  MoveL 1561 to (-1310, 1200, 50) mm, rotated rx -180 ry 0 rz 90 deg; joints [32.484, -88.139, 132.915, -62.258, 22.45, 86.682]
  MoveL 1562 to (-1310, 1200, -0.5) mm, rotated rx -180 ry 0 rz 90 deg; joints [32.484, -85.465, 133.659, -70.1, 21.066, 95.123]
  MoveL 1563 to (-1310, 1200, 50) mm, rotated rx -180 ry 0 rz 90 deg; joints [32.484, -88.139, 132.915, -62.258, 22.45, 86.682]
  MoveL 1564 to (-1380, 11.8, 50) mm, rotated rx 180 ry 0 rz 90 deg; joints [18.052, -40.759, 62.144, -21.097, 32.805, 32.18]
  MoveL 1565 to (-1380, 11.8, -0.5) mm, rotated rx 180 ry 0 rz 90 deg; joints [18.052, -39.615, 62.725, -22.113, 31.202, 33.378]
  MoveL 1566 to (-1380, 11.8, 50) mm, rotated rx 180 ry 0 rz 90 deg; joints [18.052, -40.759, 62.144, -21.097, 32.805, 32.18]
  MoveL 1567 to (-1380, 76, 50) mm, rotated rx -180 ry 0 rz 90 deg; joints [18.556, -43.766, 67.494, -23.018, 30.808, 34.667]
  MoveL 1568 to (-1380, 76, -0.5) mm, rotated rx -180 ry 0 rz 90 deg; joints [18.556, -42.567, 68.052, -24.238, 29.198, 36.076]
  MoveL 1569 to (-1380, 76, 50) mm, rotated rx -180 ry 0 rz 90 deg; joints [18.556, -43.766, 67.494, -23.018, 30.808, 34.667]
  MoveL 1570 to (-1380, 140.2, 50) mm, rotated rx 180 ry 0 rz 90 deg; joints [19.087, -46.61, 72.487, -25.083, 29.042, 37.307]
  MoveL 1571 to (-1380, 140.2, -0.5) mm, rotated rx 180 ry 0 rz 90 deg; joints [19.087, -45.356, 73.03, -26.54, 27.424, 38.96]
  MoveL 1572 to (-1380, 140.2, 50) mm, rotated rx 180 ry 0 rz 90 deg; joints [19.087, -46.61, 72.487, -25.083, 29.042, 37.307]
  MoveL 1573 to (-1450, 11.8, 50) mm, rotated rx 180 ry 0 rz 90 deg; joints [19.677, -39.594, 60.053, -22.133, 34.225, 34.119]
  MoveL 1574 to (-1450, 11.8, -0.5) mm, rotated rx -180 ry 0 rz 90 deg; joints [19.677, -38.471, 60.644, -23.132, 32.643, 35.316]
  MoveL 1575 to (-1450, 11.8, 50) mm, rotated rx 180 ry 0 rz 90 deg; joints [19.677, -39.594, 60.053, -22.133, 34.225, 34.119]
  MoveL 1576 to (-1450, 76, 50) mm, rotated rx 180 ry 0 rz 90 deg; joints [20.219, -42.64, 65.499, -24.078, 32.216, 36.683]
  MoveL 1577 to (-1450, 76, -0.5) mm, rotated rx -180 ry 0 rz 90 deg; joints [20.219, -41.462, 66.064, -25.27, 30.631, 38.08]
  MoveL 1578 to (-1450, 76, 50) mm, rotated rx 180 ry 0 rz 90 deg; joints [20.219, -42.64, 65.499, -24.078, 32.216, 36.683]
  MoveL 1579 to (-1450, 140.2, 50) mm, rotated rx 180 ry 0 rz 90 deg; joints [20.79, -45.509, 70.561, -26.153, 30.45, 39.383]
  MoveL 1580 to (-1450, 140.2, -0.5) mm, rotated rx 180 ry 0 rz 90 deg; joints [20.79, -44.276, 71.109, -27.566, 28.861, 41.009]
  MoveL 1581 to (-1450, 140.2, 50) mm, rotated rx 180 ry 0 rz 90 deg; joints [20.79, -45.509, 70.561, -26.153, 30.45, 39.383]
  MoveL 1582 to (-1520, 53.8, 50) mm, rotated rx 180 ry 0 rz 90 deg; joints [21.645, -40.349, 61.409, -24.261, 34.398, 37.539]
  MoveL 1583 to (-1520, 53.8, -0.5) mm, rotated rx 180 ry 0 rz 90 deg; joints [21.645, -39.213, 61.993, -25.347, 32.836, 38.843]
  MoveL 1584 to (-1520, 53.8, 50) mm, rotated rx 180 ry 0 rz 90 deg; joints [21.645, -40.349, 61.409, -24.261, 34.398, 37.539]
  MoveL 1585 to (-1520, 83.81, 50) mm, rotated rx 180 ry 0 rz 90 deg; joints [21.92, -41.757, 63.927, -25.195, 33.497, 38.787]
  MoveL 1586 to (-1520, 83.81, -0.5) mm, rotated rx 180 ry 0 rz 90 deg; joints [21.92, -40.595, 64.5, -26.369, 31.935, 40.183]
  MoveL 1587 to (-1520, 83.81, 50) mm, rotated rx 180 ry 0 rz 90 deg; joints [21.92, -41.757, 63.927, -25.195, 33.497, 38.787]
  MoveL 1588 to (-1520, 129.48, 50) mm, rotated rx 180 ry 0 rz 90 deg; joints [22.352, -43.823, 67.594, -26.664, 32.23, 40.736]
  MoveL 1589 to (-1520, 129.48, -0.5) mm, rotated rx 180 ry 0 rz 90 deg; joints [22.352, -42.623, 68.152, -27.983, 30.668, 42.283]
  MoveL 1590 to (-1520, 129.48, 50) mm, rotated rx 180 ry 0 rz 90 deg; joints [22.352, -43.823, 67.594, -26.664, 32.23, 40.736]
  MoveL 1591 to (-1520, 159.49, 50) mm, rotated rx 180 ry 0 rz 90 deg; joints [22.645, -45.136, 69.907, -27.661, 31.462, 42.052]
  MoveL 1592 to (-1520, 159.49, -0.5) mm, rotated rx -180 ry 0 rz 90 deg; joints [22.645, -43.911, 70.457, -29.083, 29.9, 43.705]
  MoveL 1593 to (-1520, 159.49, 50) mm, rotated rx 180 ry 0 rz 90 deg; joints [22.645, -45.136, 69.907, -27.661, 31.462, 42.052]
  MoveL 1594 to (-1520, 205.16, 50) mm, rotated rx -180 ry 0 rz 90 deg; joints [23.105, -47.076, 73.298, -29.226, 30.384, 44.107]
  MoveL 1595 to (-1520, 205.16, -0.5) mm, rotated rx -180 ry 0 rz 90 deg; joints [23.105, -45.813, 73.839, -30.815, 28.822, 45.934]
  MoveL 1596 to (-1520, 205.16, 50) mm, rotated rx -180 ry 0 rz 90 deg; joints [23.105, -47.076, 73.298, -29.226, 30.384, 44.107]
  MoveL 1597 to (-1520, 235.17, 50) mm, rotated rx 180 ry 0 rz 90 deg; joints [23.417, -48.317, 75.451, -30.286, 29.731, 45.493]
  MoveL 1598 to (-1520, 235.17, -0.5) mm, rotated rx -180 ry 0 rz 90 deg; joints [23.417, -47.029, 75.986, -31.991, 28.169, 47.441]
  MoveL 1599 to (-1520, 235.17, 50) mm, rotated rx 180 ry 0 rz 90 deg; joints [23.417, -48.317, 75.451, -30.286, 29.731, 45.493]
  MoveL 1600 to (-1520, 280.84, 50) mm, rotated rx 180 ry 0 rz 90 deg; joints [23.907, -50.16, 78.622, -31.943, 28.818, 47.655]
  MoveL 1601 to (-1520, 280.84, -0.5) mm, rotated rx 180 ry 0 rz 90 deg; joints [23.907, -48.834, 79.152, -33.836, 27.259, 49.799]
  MoveL 1602 to (-1520, 280.84, 50) mm, rotated rx 180 ry 0 rz 90 deg; joints [23.907, -50.16, 78.622, -31.943, 28.818, 47.655]
  MoveL 1603 to (-1520, 310.85, 50) mm, rotated rx -180 ry 0 rz 90 deg; joints [24.239, -51.345, 80.643, -33.06, 28.269, 49.11]
  MoveL 1604 to (-1520, 310.85, -0.5) mm, rotated rx 180 ry 0 rz 90 deg; joints [24.239, -49.994, 81.17, -35.083, 26.713, 51.39]
  MoveL 1605 to (-1520, 310.85, 50) mm, rotated rx -180 ry 0 rz 90 deg; joints [24.239, -51.345, 80.643, -33.06, 28.269, 49.11]
  MoveL 1606 to (-1520, 356.52, 50) mm, rotated rx -180 ry 0 rz 90 deg; joints [24.762, -53.113, 83.632, -34.799, 27.509, 51.372]
  MoveL 1607 to (-1520, 356.52, -0.5) mm, rotated rx -180 ry 0 rz 90 deg; joints [24.762, -51.723, 84.157, -37.029, 25.958, 53.868]
  MoveL 1608 to (-1520, 356.52, 50) mm, rotated rx -180 ry 0 rz 90 deg; joints [24.762, -53.113, 83.632, -34.799, 27.509, 51.372]
  MoveL 1609 to (-1520, 386.53, 50) mm, rotated rx -180 ry 0 rz 90 deg; joints [25.118, -54.254, 85.543, -35.963, 27.057, 52.887]
  MoveL 1610 to (-1520, 386.53, -0.5) mm, rotated rx 180 ry 0 rz 90 deg; joints [25.118, -52.838, 86.067, -38.336, 25.511, 55.533]
  MoveL 1611 to (-1520, 386.53, 50) mm, rotated rx -180 ry 0 rz 90 deg; joints [25.118, -54.254, 85.543, -35.963, 27.057, 52.887]
  MoveL 1612 to (-1690.15, 68.53, 50) mm, rotated rx -180 ry 0 rz 90 deg; joints [25.576, -37.451, 56.183, -26.136, 38.079, 41.521]
  MoveL 1613 to (-1690.15, 68.53, -0.5) mm, rotated rx 180 ry 0 rz 90 deg; joints [25.576, -36.367, 56.797, -27.135, 36.56, 42.777]
  MoveL 1614 to (-1690.15, 68.53, 50) mm, rotated rx -180 ry 0 rz 90 deg; joints [25.576, -37.451, 56.183, -26.136, 38.079, 41.521]
  MoveL 1615 to (-1690.15, 118.53, 50) mm, rotated rx -180 ry 0 rz 90 deg; joints [26.104, -39.85, 60.513, -27.686, 36.582, 43.694]
  MoveL 1616 to (-1690.15, 118.53, -0.5) mm, rotated rx 180 ry 0 rz 90 deg; joints [26.104, -38.722, 61.101, -28.811, 35.07, 45.082]
  MoveL 1617 to (-1690.15, 118.53, 50) mm, rotated rx -180 ry 0 rz 90 deg; joints [26.104, -39.85, 60.513, -27.686, 36.582, 43.694]
  MoveL 1618 to (-1690.15, 168.53, 50) mm, rotated rx 180 ry 0 rz 90 deg; joints [26.653, -42.117, 64.568, -29.281, 35.254, 45.912]
  MoveL 1619 to (-1690.15, 168.53, -0.5) mm, rotated rx -180 ry 0 rz 90 deg; joints [26.653, -40.948, 65.138, -30.543, 33.747, 47.443]
  MoveL 1620 to (-1690.15, 168.53, 50) mm, rotated rx 180 ry 0 rz 90 deg; joints [26.653, -42.117, 64.568, -29.281, 35.254, 45.912]
  MoveL 1621 to (-1690.15, 271.33, 50) mm, rotated rx -180 ry 0 rz 90 deg; joints [27.851, -46.461, 72.228, -32.698, 32.973, 50.629]
  MoveL 1622 to (-1690.15, 271.33, -0.5) mm, rotated rx 180 ry 0 rz 90 deg; joints [27.851, -45.21, 72.771, -34.268, 31.477, 52.485]
  MoveL 1623 to (-1690.15, 271.33, 50) mm, rotated rx -180 ry 0 rz 90 deg; joints [27.851, -46.461, 72.228, -32.698, 32.973, 50.629]
  MoveL 1624 to (-1690.15, 321.33, 50) mm, rotated rx -180 ry 0 rz 90 deg; joints [28.471, -48.452, 75.685, -34.418, 32.057, 52.996]
  MoveL 1625 to (-1690.15, 321.33, -0.5) mm, rotated rx 180 ry 0 rz 90 deg; joints [28.471, -47.162, 76.22, -36.152, 30.567, 55.026]
  MoveL 1626 to (-1690.15, 321.33, 50) mm, rotated rx -180 ry 0 rz 90 deg; joints [28.471, -48.452, 75.685, -34.418, 32.057, 52.996]
  MoveL 1627 to (-1690.15, 371.33, 50) mm, rotated rx -180 ry 0 rz 90 deg; joints [29.116, -50.379, 78.996, -36.168, 31.257, 55.407]
  MoveL 1628 to (-1690.15, 371.33, -0.5) mm, rotated rx -180 ry 0 rz 90 deg; joints [29.116, -49.048, 79.526, -38.073, 29.773, 57.617]
  MoveL 1629 to (-1690.15, 371.33, 50) mm, rotated rx -180 ry 0 rz 90 deg; joints [29.116, -50.379, 78.996, -36.168, 31.257, 55.407]
  MoveL 1630 to (-1566.88, 10, 50) mm, rotated rx -180 ry 0 rz 90 deg; joints [22.302, -37.259, 55.836, -23.427, 36.919, 36.788]
  MoveL 1631 to (-1566.88, 10, -0.5) mm, rotated rx 180 ry 0 rz 90 deg; joints [22.302, -36.179, 56.453, -24.369, 35.367, 37.953]
  MoveL 1632 to (-1566.88, 10, 50) mm, rotated rx -180 ry 0 rz 90 deg; joints [22.302, -37.259, 55.836, -23.427, 36.919, 36.788]
  MoveL 1633 to (-1605.08, 10, 50) mm, rotated rx 180 ry 0 rz 90 deg; joints [23.145, -36.437, 54.342, -23.771, 37.855, 37.552]
  MoveL 1634 to (-1605.08, 10, -0.5) mm, rotated rx 180 ry 0 rz 90 deg; joints [23.145, -35.371, 54.969, -24.69, 36.311, 38.704]
  MoveL 1635 to (-1605.08, 10, 50) mm, rotated rx 180 ry 0 rz 90 deg; joints [23.145, -36.437, 54.342, -23.771, 37.855, 37.552]
  MoveL 1636 to (-1643.28, 10, 50) mm, rotated rx 180 ry 0 rz 90 deg; joints [23.976, -35.567, 52.757, -24.07, 38.83, 38.253]
  MoveL 1637 to (-1643.28, 10, -0.5) mm, rotated rx -180 ry 0 rz 90 deg; joints [23.976, -34.517, 53.396, -24.965, 37.294, 39.39]
  MoveL 1638 to (-1643.28, 10, 50) mm, rotated rx 180 ry 0 rz 90 deg; joints [23.976, -35.567, 52.757, -24.07, 38.83, 38.253]
  MoveL 1639 to (-1566.88, 430, 50) mm, rotated rx 180 ry 0 rz 90 deg; joints [26.856, -55.024, 86.826, -37.945, 27.539, 56.14]
  MoveL 1640 to (-1566.88, 430, -0.5) mm, rotated rx -180 ry 0 rz 90 deg; joints [26.856, -53.59, 87.349, -40.395, 26.021, 58.885]
  MoveL 1641 to (-1566.88, 430, 50) mm, rotated rx 180 ry 0 rz 90 deg; joints [26.856, -55.024, 86.826, -37.945, 27.539, 56.14]
  MoveL 1642 to (-1605.08, 430, 50) mm, rotated rx 180 ry 0 rz 90 deg; joints [27.821, -54.295, 85.612, -38.097, 28.427, 56.884]
  MoveL 1643 to (-1605.08, 430, -0.5) mm, rotated rx -180 ry 0 rz 90 deg; joints [27.821, -52.878, 86.136, -40.439, 26.924, 59.529]
  MoveL 1644 to (-1605.08, 430, 50) mm, rotated rx 180 ry 0 rz 90 deg; joints [27.821, -54.295, 85.612, -38.097, 28.427, 56.884]
  MoveL 1645 to (-1643.28, 430, 50) mm, rotated rx -180 ry 0 rz 90 deg; joints [28.768, -53.538, 84.345, -38.194, 29.329, 57.554]
  MoveL 1646 to (-1643.28, 430, -0.5) mm, rotated rx -180 ry 0 rz 90 deg; joints [28.768, -52.138, 84.87, -40.432, 27.84, 60.102]
  MoveL 1647 to (-1643.28, 430, 50) mm, rotated rx -180 ry 0 rz 90 deg; joints [28.768, -53.538, 84.345, -38.194, 29.329, 57.554]
  MoveL 1648 to (-1520, 806.8, 50) mm, rotated rx 180 ry 0 rz 90 deg; joints [31.306, -69.147, 108.944, -52.278, 24.419, 74.949]
  MoveL 1649 to (-1520, 806.8, -0.5) mm, rotated rx 180 ry 0 rz 90 deg; joints [31.306, -67.308, 109.505, -56.727, 23.024, 79.807]
  MoveL 1650 to (-1520, 806.8, 50) mm, rotated rx 180 ry 0 rz 90 deg; joints [31.306, -69.147, 108.944, -52.278, 24.419, 74.949]
  MoveL 1651 to (-1520, 836.81, 50) mm, rotated rx 180 ry 0 rz 90 deg; joints [31.854, -70.165, 110.419, -53.283, 24.477, 76.44]
  MoveL 1652 to (-1520, 836.81, -0.5) mm, rotated rx -180 ry 0 rz 90 deg; joints [31.854, -68.291, 110.986, -57.855, 23.095, 81.435]
  MoveL 1653 to (-1520, 836.81, 50) mm, rotated rx 180 ry 0 rz 90 deg; joints [31.854, -70.165, 110.419, -53.283, 24.477, 76.44]
  MoveL 1654 to (-1520, 882.48, 50) mm, rotated rx -180 ry 0 rz 90 deg; joints [32.722, -71.711, 112.62, -54.729, 24.625, 78.65]
  MoveL 1655 to (-1520, 882.48, -0.5) mm, rotated rx -180 ry 0 rz 90 deg; joints [32.722, -69.78, 113.197, -59.473, 23.262, 83.84]
  MoveL 1656 to (-1520, 882.48, 50) mm, rotated rx -180 ry 0 rz 90 deg; joints [32.722, -71.711, 112.62, -54.729, 24.625, 78.65]
  MoveL 1657 to (-1520, 912.49, 50) mm, rotated rx 180 ry 0 rz 90 deg; joints [33.316, -72.723, 114.038, -55.618, 24.76, 80.059]
  MoveL 1658 to (-1520, 912.49, -0.5) mm, rotated rx 180 ry 0 rz 90 deg; joints [33.316, -70.755, 114.622, -60.466, 23.408, 85.367]
  MoveL 1659 to (-1520, 912.49, 50) mm, rotated rx 180 ry 0 rz 90 deg; joints [33.316, -72.723, 114.038, -55.618, 24.76, 80.059]
  MoveL 1660 to (-1520, 958.16, 50) mm, rotated rx -180 ry 0 rz 90 deg; joints [34.256, -74.262, 116.155, -56.872, 25.024, 82.129]
  MoveL 1661 to (-1520, 958.16, -0.5) mm, rotated rx 180 ry 0 rz 90 deg; joints [34.256, -72.234, 116.75, -61.861, 23.686, 87.605]
  MoveL 1662 to (-1520, 958.16, 50) mm, rotated rx -180 ry 0 rz 90 deg; joints [34.256, -74.262, 116.155, -56.872, 25.024, 82.129]
  MoveL 1663 to (-1520, 988.17, 50) mm, rotated rx 180 ry 0 rz 90 deg; joints [34.9, -75.272, 117.519, -57.625, 25.235, 83.438]
  MoveL 1664 to (-1520, 988.17, -0.5) mm, rotated rx 180 ry 0 rz 90 deg; joints [34.9, -73.203, 118.122, -62.698, 23.904, 89.015]
  MoveL 1665 to (-1520, 988.17, 50) mm, rotated rx 180 ry 0 rz 90 deg; joints [34.9, -75.272, 117.519, -57.625, 25.235, 83.438]
  MoveL 1666 to (-1520, 1033.84, 50) mm, rotated rx 180 ry 0 rz 90 deg; joints [35.922, -76.809, 119.552, -58.66, 25.612, 85.348]
  MoveL 1667 to (-1520, 1033.84, -0.5) mm, rotated rx 180 ry 0 rz 90 deg; joints [35.922, -74.676, 120.169, -63.843, 24.289, 91.063]
  MoveL 1668 to (-1520, 1033.84, 50) mm, rotated rx 180 ry 0 rz 90 deg; joints [35.922, -76.809, 119.552, -58.66, 25.612, 85.348]
  MoveL 1669 to (-1520, 1063.85, 50) mm, rotated rx 180 ry 0 rz 90 deg; joints [36.621, -77.818, 120.862, -59.264, 25.897, 86.547]
  MoveL 1670 to (-1520, 1063.85, -0.5) mm, rotated rx 180 ry 0 rz 90 deg; joints [36.621, -75.642, 121.487, -64.508, 24.576, 92.343]
  MoveL 1671 to (-1520, 1063.85, 50) mm, rotated rx 180 ry 0 rz 90 deg; joints [36.621, -77.818, 120.862, -59.264, 25.897, 86.547]
  MoveL 1672 to (-1520, 1109.52, 50) mm, rotated rx -180 ry 0 rz 90 deg; joints [37.732, -79.355, 122.812, -60.062, 26.387, 88.284]
  MoveL 1673 to (-1520, 1109.52, -0.5) mm, rotated rx -180 ry 0 rz 90 deg; joints [37.732, -77.112, 123.452, -65.385, 25.064, 94.191]
  MoveL 1674 to (-1520, 1109.52, 50) mm, rotated rx -180 ry 0 rz 90 deg; joints [37.732, -79.355, 122.812, -60.062, 26.387, 88.284]
  MoveL 1675 to (-1520, 1139.53, 50) mm, rotated rx 180 ry 0 rz 90 deg; joints [38.494, -80.366, 124.066, -60.507, 26.745, 89.368]
  MoveL 1676 to (-1520, 1139.53, -0.5) mm, rotated rx -180 ry 0 rz 90 deg; joints [38.494, -78.077, 124.716, -65.87, 25.418, 95.338]
  MoveL 1677 to (-1520, 1139.53, 50) mm, rotated rx 180 ry 0 rz 90 deg; joints [38.494, -80.366, 124.066, -60.507, 26.745, 89.368]
  MoveL 1678 to (-1690.15, 821.53, 50) mm, rotated rx 180 ry 0 rz 90 deg; joints [36.358, -65.871, 104.078, -51.46, 28.488, 77.586]
  MoveL 1679 to (-1690.15, 821.53, -0.5) mm, rotated rx -180 ry 0 rz 90 deg; joints [36.358, -64.14, 104.624, -54.915, 27.124, 81.492]
  MoveL 1680 to (-1690.15, 821.53, 50) mm, rotated rx 180 ry 0 rz 90 deg; joints [36.358, -65.871, 104.078, -51.46, 28.488, 77.586]
  MoveL 1681 to (-1690.15, 871.53, 50) mm, rotated rx 180 ry 0 rz 90 deg; joints [37.358, -67.456, 106.456, -52.866, 28.62, 79.898]
  MoveL 1682 to (-1690.15, 871.53, -0.5) mm, rotated rx 180 ry 0 rz 90 deg; joints [37.358, -65.674, 107.008, -56.456, 27.269, 83.962]
  MoveL 1683 to (-1690.15, 871.53, 50) mm, rotated rx 180 ry 0 rz 90 deg; joints [37.358, -67.456, 106.456, -52.866, 28.62, 79.898]
  MoveL 1684 to (-1690.15, 921.53, 50) mm, rotated rx 180 ry 0 rz 90 deg; joints [38.407, -69.023, 108.764, -54.167, 28.831, 82.14]
  MoveL 1685 to (-1690.15, 921.53, -0.5) mm, rotated rx -180 ry 0 rz 90 deg; joints [38.407, -67.189, 109.324, -57.879, 27.492, 86.349]
  MoveL 1686 to (-1690.15, 921.53, 50) mm, rotated rx 180 ry 0 rz 90 deg; joints [38.407, -69.023, 108.764, -54.167, 28.831, 82.14]
  MoveL 1687 to (-1690.15, 1024.33, 50) mm, rotated rx -180 ry 0 rz 90 deg; joints [40.725, -72.192, 113.297, -56.474, 29.507, 86.502]
  MoveL 1688 to (-1690.15, 1024.33, -0.5) mm, rotated rx 180 ry 0 rz 90 deg; joints [40.725, -70.244, 113.877, -60.387, 28.182, 90.969]
  MoveL 1689 to (-1690.15, 1024.33, 50) mm, rotated rx -180 ry 0 rz 90 deg; joints [40.725, -72.192, 113.297, -56.474, 29.507, 86.502]
  MoveL 1690 to (-1690.15, 1074.33, 50) mm, rotated rx -180 ry 0 rz 90 deg; joints [41.937, -73.71, 115.4, -57.401, 29.95, 88.493]
  MoveL 1691 to (-1690.15, 1074.33, -0.5) mm, rotated rx -180 ry 0 rz 90 deg; joints [41.937, -71.703, 115.992, -61.389, 28.626, 93.065]
  MoveL 1692 to (-1690.15, 1074.33, 50) mm, rotated rx -180 ry 0 rz 90 deg; joints [41.937, -73.71, 115.4, -57.401, 29.95, 88.493]
  MoveL 1693 to (-1690.15, 1124.33, 50) mm, rotated rx 180 ry 0 rz 90 deg; joints [43.21, -75.212, 117.438, -58.194, 30.465, 90.396]
  MoveL 1694 to (-1690.15, 1124.33, -0.5) mm, rotated rx 180 ry 0 rz 90 deg; joints [43.21, -73.145, 118.04, -62.24, 29.138, 95.058]
  MoveL 1695 to (-1690.15, 1124.33, 50) mm, rotated rx 180 ry 0 rz 90 deg; joints [43.21, -75.212, 117.438, -58.194, 30.465, 90.396]
  MoveL 1696 to (-1566.88, 763, 50) mm, rotated rx -180 ry 0 rz 90 deg; joints [31.883, -66.691, 105.314, -50.54, 25.501, 73.435]
  MoveL 1697 to (-1566.88, 763, -0.5) mm, rotated rx 180 ry 0 rz 90 deg; joints [31.883, -64.934, 105.863, -54.502, 24.097, 77.798]
  MoveL 1698 to (-1566.88, 763, 50) mm, rotated rx -180 ry 0 rz 90 deg; joints [31.883, -66.691, 105.314, -50.54, 25.501, 73.435]
  MoveL 1699 to (-1605.08, 763, 50) mm, rotated rx -180 ry 0 rz 90 deg; joints [32.952, -65.88, 104.092, -50.323, 26.408, 73.932]
  MoveL 1700 to (-1605.08, 763, -0.5) mm, rotated rx -180 ry 0 rz 90 deg; joints [32.952, -64.149, 104.637, -54.059, 25.012, 78.078]
  MoveL 1701 to (-1605.08, 763, 50) mm, rotated rx -180 ry 0 rz 90 deg; joints [32.952, -65.88, 104.092, -50.323, 26.408, 73.932]
  MoveL 1702 to (-1643.28, 763, 50) mm, rotated rx 180 ry 0 rz 90 deg; joints [33.997, -65.045, 102.824, -50.063, 27.318, 74.362]
  MoveL 1703 to (-1643.28, 763, -0.5) mm, rotated rx -180 ry 0 rz 90 deg; joints [33.997, -63.34, 103.366, -53.588, 25.929, 78.303]
  MoveL 1704 to (-1643.28, 763, 50) mm, rotated rx 180 ry 0 rz 90 deg; joints [33.997, -65.045, 102.824, -50.063, 27.318, 74.362]
  MoveL 1705 to (-1566.88, 1183, 50) mm, rotated rx 180 ry 0 rz 90 deg; joints [41.145, -80.512, 124.245, -60.536, 28.397, 91.467]
  MoveL 1706 to (-1566.88, 1183, -0.5) mm, rotated rx -180 ry 0 rz 90 deg; joints [41.145, -78.215, 124.896, -65.537, 27.059, 97.116]
  MoveL 1707 to (-1566.88, 1183, 50) mm, rotated rx 180 ry 0 rz 90 deg; joints [41.145, -80.512, 124.245, -60.536, 28.397, 91.467]
  MoveL 1708 to (-1605.08, 1183, 50) mm, rotated rx -180 ry 0 rz 90 deg; joints [42.319, -79.422, 122.895, -60.081, 29.264, 91.873]
  MoveL 1709 to (-1605.08, 1183, -0.5) mm, rotated rx 180 ry 0 rz 90 deg; joints [42.319, -77.175, 123.535, -64.778, 27.927, 97.221]
  MoveL 1710 to (-1605.08, 1183, 50) mm, rotated rx -180 ry 0 rz 90 deg; joints [42.319, -79.422, 122.895, -60.081, 29.264, 91.873]
  MoveL 1711 to (-1643.28, 1183, 50) mm, rotated rx 180 ry 0 rz 90 deg; joints [43.451, -78.32, 121.504, -59.591, 30.122, 92.203]
  MoveL 1712 to (-1643.28, 1183, -0.5) mm, rotated rx -180 ry 0 rz 90 deg; joints [43.451, -76.123, 122.134, -64.006, 28.784, 97.272]
  MoveL 1713 to (-1643.28, 1183, 50) mm, rotated rx 180 ry 0 rz 90 deg; joints [43.451, -78.32, 121.504, -59.591, 30.122, 92.203]
  Set speed (1000.0 mm/s)
  MoveL 1714 to (-1643.28, 1183, 50) mm, rotated rx 180 ry 0 rz 90 deg; joints [43.451, -78.32, 121.504, -59.591, 30.122, 92.203]
  MoveL 1715 to (-1643.28, 1183, 150) mm, rotated rx -180 ry 0 rz 90 deg; joints [43.451, -82.307, 119.902, -52.09, 33.269, 83.395]
